{attribute addProperty BoxType "EK1122-0000-0018"}
{attribute addProperty Id "Beckhoff_CUxxxxsub_EK1100EK1100_179A0949162A_0001_CU1123_0000_0016A_0001_CU1123_0000_0016_6E4C53AF992124"}
{attribute addProperty CRC "1094630127"}
{attribute addProperty SizeInBites "1008"}
{attribute addProperty SizeInBytes "126"}
TYPE Beckhoff_CUxxxxEK1122_413EBAEF EXTENDS EK1122_179A0949 :
STRUCT
	{attribute addProperty Name "Beckhoff_CUxxxxsub_EK1100"}
	Beckhoff_CUxxxxsub_EK1100 : EK1100_179A0949;
	{attribute addProperty Name "A_0001_CU1123_0000_0016"}
	A_0001_CU1123_0000_0016 : A_0001_CU1123_0000_0016_6E4C53AF;
END_STRUCT
END_TYPE

(* stored: Version 1.2.0.0, ProductVersion 3.1.4024.9
   DUT Beckhoff_CUxxxxEK1122_413EBAEF: Id {c320d9b7-58b3-49f7-a309-723e88d55e3f} *)
